Staubli VAL3: motion_cntl.pgx

public program motion_cntl()
begin

  do

    wait(spd_cntl == true)
    setMonitorSpeed(Ref_Vel)

  until check_status != true

end
